{attribute 'linkalways'} 
{attribute 'no_explicit_call' := 'This FB is a CLASS and must be accessed using methods or properties'}
{attribute 'enable_dynamic_creation'}
FUNCTION_BLOCK Node_F_VN_BrightBorderObjects EXTENDS VisionNode
VAR
    ipSrcImage : _ITcVnImage;
    ipDestImage : _ITcVnImage;
    hrPrev : _HRESULT(S_OK);
	hresult : _HRESULT(S_OK);
END_VAR

METHOD PUBLIC  Clone : I_Node
VAR
	pNode : POINTER TO Node_F_VN_BrightBorderObjects;
END_VAR
pNode := __NEW(Node_F_VN_BrightBorderObjects);
Clone := pNode^;
END_METHOD

METHOD FB_init : BOOL
VAR_INPUT
	bInitRetains : BOOL; // if TRUE, the retain variables are initialized (warm start / cold start)
	bInCopyCode : BOOL;  // if TRUE, the instance afterwards gets moved into the copy code (online change)
END_VAR
AddInput('ipSrcImage', ipSrcImage);
AddInput('hrPrev', hrPrev);
AddOutput('ipDestImage', ipDestImage);
AddOutput('hresult',hresult);
END_METHOD

METHOD PROTECTED OnExecute : HRESULT
hresult.Value := F_VN_BrightBorderObjects(
    ipSrcImage := ipSrcImage.Value,
	ipDestImage := ipDestImage.Value,
	hrPrev:= hrPrev.Value);
END_METHOD

METHOD PUBLIC PreExecutionCheck
VAR_INPUT
	Check : I_PreExecutionChecks;
END_VAR
IF FAILED(hrPrev.Value) THEN
    RETURN;
END_IF

Check.IsTrue(ipSrcImage.IsValid, 'ipSrcImage must contain an image');
Check.IsTrue(ipSrcImage.HasChannelCount(1), 'ipSrcImage must have 1 channel');

Check.IsTrue((ipSrcImage.IsPixelDepth(8)  OR
              ipSrcImage.IsPixelDepth(16) OR
              ipSrcImage.IsPixelDepth(32) OR
              ipSrcImage.IsPixelDepth(64)), 'ipSrcImage must have 8, 16, 32 or 64 bit pixel depth');
END_METHOD

END_FUNCTION_BLOCK

(* stored: Version 1.1.0.1, ProductVersion 3.1.4024.13
   POU Node_F_VN_BrightBorderObjects: Id {031eaaa9-1dd6-0a55-2786-61a7633985e3}, SpecialFunc None
   Folder Constructor: Id {a88c26c9-91b4-0119-04f9-9fbe73365998}
   Method Clone: Id {b29986ad-0e28-03d2-2504-68d8182b020e}
   Method FB_init: Id {1913c3db-ccd8-01a8-3bcf-bbcba75aa0b7}
   Method OnExecute: Id {c676fffd-51d2-0812-2573-fdb0ff080cd5}
   Method PreExecutionCheck: Id {f6c647ec-8195-0f7a-2efd-1e010aef0f69} *)
